FUNCTION_BLOCK FB_LamparaAsignada_SFC
// La lampara se enciende mientras se acciona el pulsador
VAR
    Lampara   AT %Q*  : BOOL;
    Pulsador  AT %I*  : BOOL;
END_VAR

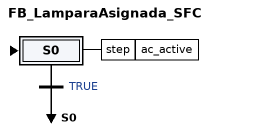
INITIAL_STEP S0:
    ac_active(N);  // step action
END_STEP
TRANSITION FROM S0 TO S0
    := TRUE;
END_TRANSITION

ACTION ac_active:
Lampara := S0.x AND Pulsador;
END_ACTION

END_FUNCTION_BLOCK

(* stored: Version 1.1.0.1, ProductVersion 3.1.4024.15
   POU FB_LamparaAsignada_SFC: Id {4accafcd-bc48-433a-ace9-cfe04d71a8e2}, SpecialFunc None
   Action ac_active: Id {cff54ff1-6796-45ab-9e03-7da13421d66e} *)
